// TIA Portal V17 export
// export: Created 2025-03-05T08:00:15.229314Z, ExportSetting WithDefaults, DisplayName Totally Integrated Automation Portal, DisplayVersion V17 Update 8, DisplayName TIA Portal Openness, DisplayVersion V17 Update 8, DisplayName TIA Portal Version Control Interface, DisplayVersion V17, DisplayName SINAMICS Startdrive Advanced, DisplayVersion V17 SP2, DisplayName SINAMICS Startdrive G110M, G120, G120C, G120D, G120P, G115D, DisplayVersion V17 SP2, DisplayName SINAMICS Startdrive G130, G150, S120, S150, SINAMICS MV, S210, DisplayVersion V17 SP2, DisplayName STEP 7 Professional, DisplayVersion V17 Update 8, DisplayName SINUMERIK ONE STEP 7 Toolbox, DisplayVersion V17 Update 12, DisplayName SINUMERIK 840D sl STEP 7 Toolbox, DisplayVersion V17 Update 12, DisplayName STEP 7 Safety, DisplayVersion V17 Update 6, DisplayName WinCC Advanced, DisplayVersion V17 Update 8
DATA_BLOCK "DB2101_LINE_CONTACTOR"   // DB2101
{ S7_Optimized_Access := 'FALSE'; DB_Accessible_From_OPC_UA := 'FALSE' }
AUTHOR : ETXETAR
VERSION : 1.0
// stored: AutoNumber false, DBAccessibleFromOPCUA false, DBAccessibleFromWebserver true, IsOnlyStoredInLoadMemory false, IsWriteProtectedInAS false
   VAR
      FEEDBACK_IN_1 : Bool;   // CONTACTOR FEEDBACK INPUT 1
      FEEDBACK_IN_2 : Bool;   // CONTACTOR FEEDBACK INPUT 2
      LINE_CONTACTOR_ENABLED : Bool;   // LINE CONTACTOR ENABLED
      ON_GENERAL_CONDITIONS : Bool;   // UNIT 01L CYCLE SEQUENCE GENERAL CONDITIONS / SWITCH ON GENERAL CONDITIONS
      ON_INITIAL_CONDITIONS : Bool;   // UNIT 01L CYCLE SEQUENCE INITIAL CONDITIONS / SWITCH ON INITIAL CONDITIONS
      ON_REQ_1 : Bool;   // UNIT 01L CYCLE SEQUENCE STEP 4 / SWITCH ON REQUEST 1
      ON_REQ_2 : Bool;   // UNIT 01L CYCLE SEQUENCE STEP 5 / SWITCH ON REQUEST 2
      ON_REQ_3 : Bool;   // UNIT 01L CYCLE SEQUENCE STEP 6 / SWITCH ON REQUEST 3
      ON_REQ_4 : Bool;   // UNIT 01L CYCLE SEQUENCE STEP 7 / SWITCH ON REQUEST 4
      OFF_GENERAL_CONDITIONS : Bool;   // UNIT 01L CYCLE SEQUENCE GENERAL CONDITIONS / SWITCH OFF GENERAL CONDITIONS
      OFF_INITIAL_CONDITIONS : Bool;   // UNIT 01L CYCLE SEQUENCE INITIAL CONDITIONS / SWITCH OFF INITIAL CONDITIONS
      OFF_REQ_1 : Bool;   // UNIT 01L CYCLE SEQUENCE STEP 4 / SWITCH OFF REQUEST 1
      OFF_REQ_2 : Bool;   // UNIT 01L CYCLE SEQUENCE STEP 5 / SWITCH OFF REQUEST 2
      OFF_REQ_3 : Bool;   // UNIT 01L CYCLE SEQUENCE STEP 6 / SWITCH OFF REQUEST 3
      OFF_REQ_4 : Bool;   // UNIT 01L CYCLE SEQUENCE STEP 7 / SWITCH OFF REQUEST 4
      STEP_1_CONTACTOR_ON : Bool;   // UNIT 01L CYCLE SEQUENCE STEP 1 / STEP 1
      STEP_2_POWER_SUPPLY_ON : Bool;   // UNIT 01L CYCLE SEQUENCE STEP 2 / STEP 2
      STEP_3_OFF3_ON : Bool;   // UNIT 01L CYCLE SEQUENCE STEP 3 / STEP 3
      STEP_4 : Bool;   // UNIT 01L CYCLE SEQUENCE STEP 8 / STEP 4
      STEP_5 : Bool;   // UNIT 01L CYCLE SEQUENCE STEP 9 / STEP 5
      STEP_6 : Bool;   // UNIT 01L CYCLE SEQUENCE STEP 10 / STEP 6
      STEP_7 : Bool;   // UNIT 01L CYCLE SEQUENCE STEP 11 / STEP 7
      FEEDBACK_1_ALM : Bool;   // CONTACTOR FEEDBACK 1 ALARM
      FEEDBACK_2_ALM : Bool;   // CONTACTOR FEEDBACK 2 ALARM
      O_LINE_CONTACTOR_1 : Bool;   // UNIT 01L CYCLE SEQUENCE AUX0 / OPTION LINE CONTACTOR 1
      O_LINE_CONTACTOR_2 : Bool;   // UNIT 01L CYCLE SEQUENCE AUX1 / OPTION LINE CONTACTOR 2
      AUX2 : Bool;   // UNIT 01L CYCLE SEQUENCE AUX2 / AUXILIARY 2
      AUX3 : Bool;   // UNIT 01L CYCLE SEQUENCE AUX3 / AUXILIARY 3
      AUX5 : Bool;   // UNIT 01L CYCLE SEQUENCE AUX5 / AUXILIARY 5
      AUX6 : Bool;   // UNIT 01L CYCLE SEQUENCE AUX6 / AUXILIARY 6
      AUX7 : Bool;   // UNIT 01L CYCLE SEQUENCE AUX7 / AUXILIARY 7
      AUX8 : Bool;   // UNIT 01L CYCLE SEQUENCE AUX7 / AUXILIARY 8
      NOT_SWITCHED_ON_WARNING : Bool;   // LINE CONTACTOR NOT SWITCHED ON WARNING
      GENERAL_CONDITIONS_HELP : Bool;   // UNIT 01L CYCLE SEQUENCE GENERAL CONDITIONS HELP / GENERAL CONDITIONS HELP
      INITIAL_CONDITIONS_HELP : Bool;   // UNIT 01L CYCLE SEQUENCE INITIAL CONDITIONS HELP / INITIAL CONDITIONS HELP
      ANY_ACTIVE_ALARM : Bool;   // ANY ACTIVE ALARM
      IS_ALARMS : Bool;   // IMMEDIATE STOP ALARMS
      WARNINGS : Bool;   // WARNINGS
      WARNINGS_GONE : Bool;   // UNIT 01L CYCLE SEQUENCE PREALARM GONE / WARNINGS GONE
      TIMER_CONTACTOR_LINE_FEEDBACK_1 : TON_TIME;   // CONTACTOR LINE FEEDBACK 1 TIMER
      TIMER_CONTACTOR_LINE_FEEDBACK_2 : TON_TIME;   // CONTACTOR LINE FEEDBACK 2 TIMER
      TIMER_STEP_2_START_ON : TON_TIME;   // STEP 1 START ON TIMER
      TIMER_STEP_3_START_ON : TON_TIME;   // STEP 2 START ON TIMER
      TIMER_EMERGENCY_STOP_PILZ_REQUEST : TON_TIME;   // EMERGENCY STOP PILZ REQUEST TIMER
      TIMER_START_OFF_REQUEST_2 : TOF_TIME;   // START OFF REQUEST 1 TIMER
      TIMER_START_OFF_REQUEST_3 : TOF_TIME;   // START OFF REQUEST 2 TIMER
   END_VAR
BEGIN
   TIMER_CONTACTOR_LINE_FEEDBACK_1.PT := T#500ms;
   TIMER_CONTACTOR_LINE_FEEDBACK_2.PT := T#500ms;
   TIMER_STEP_2_START_ON.PT := T#1s;
   TIMER_STEP_3_START_ON.PT := T#100ms;
   TIMER_EMERGENCY_STOP_PILZ_REQUEST.PT := T#5s;
   TIMER_START_OFF_REQUEST_2.PT := T#1s;
   TIMER_START_OFF_REQUEST_3.PT := T#1s;
END_DATA_BLOCK
